FUNCTION_BLOCK LevitationEqualizingController
VAR_INPUT
	// Actual delta F value
	fActualdF : LREAL;
END_VAR

VAR
	// PID function block	
	fbPID : FB_BasicPID;
	// PID parameters
	fSetpointValue : LREAL;
	bReset : BOOL;
	fCtrlCycleTime : LREAL;
	fKp : LREAL;
	fTn : LREAL;
	fTv : LREAL;
	fTd : LREAL;
	// PID outputs	
	fCtrlOutput : LREAL;
	// Saturation parameter
	fdzMax : LREAL := 0.001;
	fdzMin : LREAL := -0.001;
END_VAR
VAR_OUTPUT
	// dz output vector
	fdz : ARRAY[1..4] OF LREAL;
	nErrorStatus : UINT;
END_VAR

fbPID(fSetpointValue := fSetpointValue,
	  fActualValue := fActualdF,
	  bReset := bReset,
	  fCtrlCycleTime := fCtrlCycleTime,
	  fKp := fKp,
	  fTn := fTn,
	  fTv := fTv,
	  fTd := fTd,
	  fCtrlOutput => fCtrlOutput, nErrorStatus => nErrorStatus);
	  
// Update the dz output vector
fdz[1] := -1/7900*fCtrlOutput; // TO DO : change it to lookup table function F_inv(F)
fdz[2] := 1/7900*fCtrlOutput;
fdz[3] := -1/7900*fCtrlOutput;
fdz[4] := 1/7900*fCtrlOutput;	  

// Saturate the dz output vector
IF fdz[1] > fdzMax THEN
	fdz[1] := fdzMax;
ELSIF fdz[1] < fdzMin THEN
	fdz[1] := fdzMin;
END_IF

IF fdz[2] > fdzMax THEN
	fdz[2] := fdzMax;
ELSIF fdz[2] < fdzMin THEN
	fdz[2] := fdzMin;
END_IF

IF fdz[3] > fdzMax THEN
	fdz[3] := fdzMax;
ELSIF fdz[3] < fdzMin THEN
	fdz[3] := fdzMin;
END_IF

IF fdz[4] > fdzMax THEN
	fdz[4] := fdzMax;
ELSIF fdz[4] < fdzMin THEN
	fdz[4] := fdzMin;
END_IF

METHOD FB_init : BOOL
VAR_INPUT
	bInitRetains : BOOL; // if TRUE, the retain variables are initialized (warm start / cold start)
	bInCopyCode : BOOL;  // if TRUE, the instance afterwards gets moved into the copy code (online change)
	fSetpointValue : LREAL;
	bReset : BOOL;
	fCtrlCycleTime : LREAL;
	fKp : LREAL;
	fTn : LREAL;
	fTv : LREAL;
	fTd : LREAL;
END_VAR
THIS^.fSetpointValue := fSetpointValue;
THIS^.bReset := bReset;
THIS^.fCtrlCycleTime := fCtrlCycleTime;
THIS^.fKp := fKp;
THIS^.fTn := fTn;
THIS^.fTv := fTv;
THIS^.fTd := fTd;
END_METHOD

END_FUNCTION_BLOCK

(* stored: Version 1.1.0.1, ProductVersion 3.1.4024.12
   POU LevitationEqualizingController: Id {bf86a80d-a85a-47bc-a5bf-df6659343b99}, SpecialFunc None
   Method FB_init: Id {482ee31a-e300-4819-9a24-f26f4af1074f} *)
